// TIA Portal V20 export
DATA_BLOCK "SomeInstance"   // DB4
// stored: InstanceOfName SomeFB, InstanceOfType FB
"SomeFB"
   // VAR_INPUT
   //    InWord0 : Word;
   // END_VAR
   // VAR_OUTPUT
   //    OutWord0 : Word;
   // END_VAR
   // VAR
   //    Flag : Bool;
   // END_VAR
BEGIN
END_DATA_BLOCK
